{attribute 'linkalways'} 
{attribute 'no_explicit_call' := 'This FB is a CLASS and must be accessed using methods or properties'}
{attribute 'enable_dynamic_creation'}
FUNCTION_BLOCK FINAL MOD_DWORD EXTENDS Node
VAR
	in1 : _DWORD(0);
	in2 : _DWORD(0);
	out : _DWORD(0);
END_VAR

METHOD PUBLIC Clone : I_Node
VAR
	pNode : POINTER TO MOD_DWORD;
END_VAR
pNode := __NEW(MOD_DWORD);
Clone := pNode^;
END_METHOD

METHOD FB_init : BOOL
VAR_INPUT
	bInitRetains : BOOL; // if TRUE, the retain variables are initialized (warm start / cold start)
	bInCopyCode : BOOL;  // if TRUE, the instance afterwards gets moved into the copy code (online change)
END_VAR
AddInput('in1',THIS^.in1);
AddInput('in2',THIS^.in2);
AddOutput('out', THIS^.out);
END_METHOD

METHOD PROTECTED OnExecute
VAR
END_VAR
out.Value := in1.Value MOD in2.Value;
END_METHOD

END_FUNCTION_BLOCK

(* stored: Version 1.1.0.1, ProductVersion 3.1.4024.15
   POU MOD_DWORD: Id {40c35c96-d852-456d-8d95-aaef188f0e89}, SpecialFunc None
   Folder Constructor: Id {9366af1e-4624-41e4-9312-a8e2f3ec17ef}
   Method Clone: Id {de30efc9-87fb-4e40-be6f-15119901d9d1}
   Method FB_init: Id {f859a78c-375b-4a49-a98c-e6f1c4b95b97}
   Method OnExecute: Id {18b796fb-c34f-40f5-abab-02eb0412e7a9} *)
